INTERFACE I_Navitrol_StreamVelocity EXTENDS I_Base, I_Enablable, I_TaskResult

METHOD SetTargetVelocity
VAR_INPUT
	TargetVelocity : LREAL; // Desired velocity setpoint (signed)
END_VAR
END_METHOD

END_INTERFACE

(* stored: Version 1.1.0.1
   Itf I_Navitrol_StreamVelocity: Id {4162c3a6-8f05-4586-adcf-ada9b9a3278a}
   Method SetTargetVelocity: Id {c2ab01a1-a632-43a4-b9c5-d59ed81e2c02} *)
